INTERFACE IUnitTest EXTENDS __SYSTEM.IQueryInterface

METHOD Execute
END_METHOD

METHOD Initialise
VAR_INPUT
    MessageList : IAssertionMessageList;
END_VAR
END_METHOD

PROPERTY TestHasFailed : BOOL
GET
END_GET
END_PROPERTY

PROPERTY TestHasFinished : BOOL
GET
END_GET
END_PROPERTY

PROPERTY TestName : T_MaxString
GET
END_GET
END_PROPERTY

END_INTERFACE

(* stored: Version 1.1.0.1, ProductVersion 3.1.4024.3
   Itf IUnitTest: Id {5e460ea2-01bf-4593-869c-becd2e132076}
   Method Execute: Id {00e9f158-bca0-4be7-a174-a15e36fcc65a}
   Method Initialise: Id {cd64242e-1f32-4ced-9d69-d4b7ba086760}
   Property TestHasFailed: Id {854419ed-e6e4-4501-9739-9f2599603c49}
   Get Get: Id {501edbb7-2012-47d9-9084-a3a726be116b}
   Property TestHasFinished: Id {3d152a58-6272-4064-abb2-eeebd29a939a}
   Get Get: Id {7c8499ab-f5ef-4220-a14d-ad19cc7feb49}
   Property TestName: Id {c0200cb1-9a92-421b-9ae6-b7096513949b}
   Get Get: Id {b5f54003-5f0e-4749-b3c4-d14fcadd532f} *)
